PROGRAM RunToTarget
VAR
	ClearToRun	: BOOL := FALSE;
	TargetClear	: BOOL := HMI.bTgtLoaded;
	CurrentPos	: REAL := XML.savedvalues.CurrentPos;
	TargetPos	: REAL := GV_HMI.TargetPos;
	UpLim		: REAL := XML.savedvalues.FwdSoftLim;
	DwnLim		: REAL := XML.savedvalues.RevSoftLim;
	TargetTol	: REAL := 0.25;
	UpToL		: REAL := TargetPos + TargetTol;
	DownTol		: REAL := TargetPos - TargetTol;
	UpEnable	: BOOL := FALSE;
	DownEnable	: BOOL := FALSE;
END_VAR

//Determines if System is Clear to Run
	IF CurrentPos > UpLim 

//Run to Position Enabling
	//Runs UP to Position
		IF CleartoRun = TRUE AND CurrentPos > TargetPos THEN
			UpEnable := TRUE;
	//Runs DOWN to Position	
		ELSIF ClearToRun = TRUE AND CurrentPos < TargetPos THEN
			DownEnable := TRUE;
		END_IF
		
//

END_PROGRAM

(* stored: Version 1.1.0.1, ProductVersion 3.1.4022.12
   POU RunToTarget: Id {5a6b594f-be09-44db-803b-53b32e0cebfb}, SpecialFunc None *)
